{attribute 'qualified_only'}
//{attribute 'strict'}
TYPE eModemState :
(
	Disconnected := 0,
	Connected := 1
);
END_TYPE

(* stored: Version 1.1.0.1, ProductVersion 3.1.4026.18
   DUT eModemState: Id {3c275668-523d-458d-832b-02adfc587bb8} *)
